FUNCTION_BLOCK ProfiNetDeviceBase
VAR_INPUT
END_VAR
VAR_OUTPUT
END_VAR
VAR
	PnIoDeviceState AT%I* : UINT;
	PnIoDeviceDiag AT%i* : uint;
END_VAR

END_FUNCTION_BLOCK

(* stored: Version 1.1.0.1, ProductVersion 3.1.4024.11
   POU ProfiNetDeviceBase: Id {c9b78d03-7160-4d15-a463-d097735815ac}, SpecialFunc None *)
